TYPE ST_PneumaticAxisStruct :
STRUCT
    stPneumaticAxisInputs: ST_PneumaticAxisInputs;
    stPneumaticAxisOutputs: ST_PneumaticAxisOutputs;
    stPneumaticAxisControl: ST_PneumaticAxisControl;
    stPneumaticAxisStatus: ST_PneumaticAxisStatus;
    stPneumaticAxisConfig: ST_PneumaticAxisConfig;
    ePneumaticAxisMode: E_PneumaticMode;
    ePneumaticAxisErrors: E_PneumaticAxisErrors;
END_STRUCT
END_TYPE

(* stored: Version 1.1.0.1, ProductVersion 3.1.4024.12
   DUT ST_PneumaticAxisStruct: Id {d6160476-b349-4ae7-92a0-2b29d5177a8e} *)
